{attribute 'qualified_only'}
VAR_GLOBAL
END_VAR

(* stored: Version 1.1.0.1, ProductVersion 3.1.4024.12
   GVL G_Parameters: Id {2bd5be29-f937-4001-8bc0-48e574ea2054} *)
